// TIA Portal V19 export
VAR_GLOBAL   // PLC tag table "Speed Control"
   POT2_Lower_Real AT %MD38 : Real;
   Tmp AT %MW4 : Word;
   POT1_Upper__Real AT %MD16 : Real;
   MyIndex AT %MW6 : Int;
   Drive_Error AT %M11.3 : Bool;
   OS2 AT %M10.3 : Bool;
   OS3 AT %M10.5 : Bool;
   G120_Error AT %M10.6 : Bool;
   G120_Enabled AT %M10.7 : Bool;
   G120_Run_Velocity AT %M11.0 : Bool;
   OS4 AT %M11.1 : Bool;
   OS5 AT %M11.2 : Bool;
   BusyMV AT %M0.0 : Bool;
END_VAR
